// TIA Portal V20 export
ORGANIZATION_BLOCK "Main"   // OB128, LAD, ProgramCycle
TITLE = "Main Program Sweep (Cycle)"
// stored: Namespace CITI_Logic, SetENOAutomatically false
   VAR_INPUT
      Initial_Call : Bool;   // Initial call of this OB
      Remanence : Bool;   // =True, if remanent data are available
   END_VAR
   VAR_TEMP
      tempEnable : Bool;   // Replace with the user tags
      tempFilter : Bool;   // Replace with the user tags
      tempValid : Bool;   // Replace with the user tags
      tempBusy : Bool;   // Replace with the user tags
      tempError : Bool;   // Replace with the user tags
      tempStatus : Word;   // Replace with the user tags
   END_VAR
   VAR_TEMP   // added for the SCL form of the ladder/FBD networks
      _w1 : Bool;
   END_VAR
BEGIN

REGION Network 1
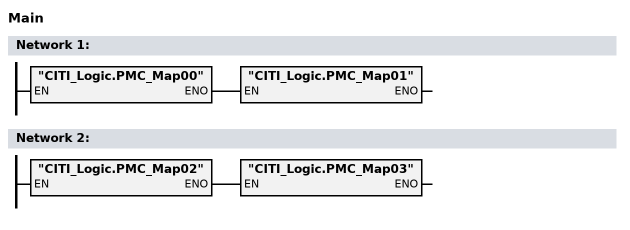
   RUNG wire#powerrail
      "CITI_Logic.PMC_Map00"()
      "CITI_Logic.PMC_Map01"()
   END_RUNG
   // the same network as SCL:
   "CITI_Logic.PMC_Map00"(ENO => #_w1);
   IF #_w1 THEN "CITI_Logic.PMC_Map01"(); END_IF;
END_REGION

REGION Network 2
   RUNG wire#powerrail
      "CITI_Logic.PMC_Map02"()
      "CITI_Logic.PMC_Map03"()
   END_RUNG
   // the same network as SCL:
   "CITI_Logic.PMC_Map02"(ENO => #_w1);
   IF #_w1 THEN "CITI_Logic.PMC_Map03"(); END_IF;
END_REGION
END_ORGANIZATION_BLOCK
